ABB RobotStudio station: Solution14.rsstn

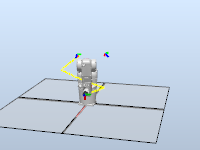
Station Solution14 (saved by RobotStudio 21.4.9700.0)
Controller IRB1200_7_70
  mechanical unit ROB_1: IRB1200_7_70_STD_03, 6 joints, base frame (0, 0, 0) mm
Layout (positions relative to the parent item):
  - IRB1200_7_70_STD_03 [mechanism, from Robots\IRB1200_7_70_STD_03.rslib] at (0, 0, 0) mm; joint values [0.2477, 0.9851, 0.7667, 0.2515, -1.7464, 0.0449] (rad or m)
Targets, tools, work objects and paths stored in the station, written as RAPID:
! task T_ROB1
MODULE Module1
  CONST robtarget Target_10:=[[422.01408311,0,750.1],[0.5,0,0.866025404,0],[0,0,0,0],[9E+09,9E+09,9E+09,9E+09,9E+09,9E+09]];
  CONST robtarget Target_20:=[[291.100367613,305.542897674,750.1],[0.459590616,-0.341070954,0.796034298,0.196917407],[0,0,-1,0],[9E+09,9E+09,9E+09,9E+09,9E+09,9E+09]];
  CONST jointtarget JointTarget_0:=[[-1.2,-19.89,29.46,-7.2,-9.64,7.1],[9E+09,9E+09,9E+09,9E+09,9E+09,9E+09]];
  CONST jointtarget JointTarget_1:=[[-2.4,-19.76,29.97,-13.32,-10.49,13.1],[9E+09,9E+09,9E+09,9E+09,9E+09,9E+09]];
  CONST jointtarget JointTarget_2:=[[-3.6,-19.59,30.47,-18.45,-11.45,18.1],[9E+09,9E+09,9E+09,9E+09,9E+09,9E+09]];
  CONST jointtarget JointTarget_3:=[[-4.79,-19.41,30.95,-22.74,-12.49,22.26],[9E+09,9E+09,9E+09,9E+09,9E+09,9E+09]];
  CONST jointtarget JointTarget_4:=[[-5.98,-19.2,31.42,-26.34,-13.59,25.69],[9E+09,9E+09,9E+09,9E+09,9E+09,9E+09]];
  CONST jointtarget JointTarget_5:=[[-7.17,-18.97,31.88,-29.36,-14.74,28.55],[9E+09,9E+09,9E+09,9E+09,9E+09,9E+09]];
  CONST jointtarget JointTarget_6:=[[-8.34,-18.72,32.33,-31.92,-15.92,30.93],[9E+09,9E+09,9E+09,9E+09,9E+09,9E+09]];
  CONST jointtarget JointTarget_7:=[[-9.51,-18.44,32.76,-34.11,-17.14,32.91],[9E+09,9E+09,9E+09,9E+09,9E+09,9E+09]];
  CONST jointtarget JointTarget_8:=[[-10.67,-18.14,33.17,-35.98,-18.37,34.57],[9E+09,9E+09,9E+09,9E+09,9E+09,9E+09]];
  CONST jointtarget JointTarget_9:=[[-11.82,-17.81,33.58,-37.61,-19.61,35.96],[9E+09,9E+09,9E+09,9E+09,9E+09,9E+09]];
  CONST jointtarget JointTarget_11:=[[-14.09,-17.09,34.33,-40.25,-22.13,38.1],[9E+09,9E+09,9E+09,9E+09,9E+09,9E+09]];
  CONST jointtarget JointTarget_12:=[[-15.21,-16.69,34.69,-41.34,-23.4,38.92],[9E+09,9E+09,9E+09,9E+09,9E+09,9E+09]];
  CONST jointtarget JointTarget_13:=[[-16.31,-16.27,35.03,-42.3,-24.66,39.59],[9E+09,9E+09,9E+09,9E+09,9E+09,9E+09]];
  CONST jointtarget JointTarget_14:=[[-17.4,-15.83,35.36,-43.16,-25.93,40.14],[9E+09,9E+09,9E+09,9E+09,9E+09,9E+09]];
  CONST jointtarget JointTarget_15:=[[-18.48,-15.37,35.67,-43.93,-27.19,40.6],[9E+09,9E+09,9E+09,9E+09,9E+09,9E+09]];
  CONST jointtarget JointTarget_16:=[[-19.55,-14.89,35.97,-44.63,-28.44,40.95],[9E+09,9E+09,9E+09,9E+09,9E+09,9E+09]];
  CONST jointtarget JointTarget_17:=[[-20.59,-14.38,36.24,-45.25,-29.69,41.23],[9E+09,9E+09,9E+09,9E+09,9E+09,9E+09]];
  CONST jointtarget JointTarget_18:=[[-21.63,-13.85,36.51,-45.83,-30.92,41.44],[9E+09,9E+09,9E+09,9E+09,9E+09,9E+09]];
  CONST jointtarget JointTarget_19:=[[-22.65,-13.3,36.75,-46.35,-32.15,41.59],[9E+09,9E+09,9E+09,9E+09,9E+09,9E+09]];
  CONST jointtarget JointTarget_21:=[[-24.64,-12.14,37.2,-47.28,-34.58,41.72],[9E+09,9E+09,9E+09,9E+09,9E+09,9E+09]];
  CONST jointtarget JointTarget_22:=[[-25.61,-11.53,37.4,-47.7,-35.77,41.72],[9E+09,9E+09,9E+09,9E+09,9E+09,9E+09]];
  CONST jointtarget JointTarget_23:=[[-26.57,-10.9,37.58,-48.09,-36.95,41.68],[9E+09,9E+09,9E+09,9E+09,9E+09,9E+09]];
  CONST jointtarget JointTarget_24:=[[-27.51,-10.26,37.74,-48.45,-38.11,41.6],[9E+09,9E+09,9E+09,9E+09,9E+09,9E+09]];
  CONST jointtarget JointTarget_25:=[[-28.43,-9.59,37.89,-48.8,-39.26,41.49],[9E+09,9E+09,9E+09,9E+09,9E+09,9E+09]];
  CONST jointtarget JointTarget_26:=[[-29.34,-8.91,38.02,-49.13,-40.39,41.35],[9E+09,9E+09,9E+09,9E+09,9E+09,9E+09]];
  CONST jointtarget JointTarget_27:=[[-30.23,-8.21,38.13,-49.44,-41.51,41.19],[9E+09,9E+09,9E+09,9E+09,9E+09,9E+09]];
  CONST jointtarget JointTarget_28:=[[-31.1,-7.5,38.22,-49.74,-42.6,41],[9E+09,9E+09,9E+09,9E+09,9E+09,9E+09]];
  CONST jointtarget JointTarget_29:=[[-31.96,-6.77,38.3,-50.03,-43.68,40.79],[9E+09,9E+09,9E+09,9E+09,9E+09,9E+09]];
  CONST jointtarget JointTarget_30:=[[-32.8,-6.03,38.36,-50.32,-44.75,40.56],[9E+09,9E+09,9E+09,9E+09,9E+09,9E+09]];
  CONST jointtarget JointTarget_31:=[[-33.63,-5.27,38.4,-50.59,-45.79,40.32],[9E+09,9E+09,9E+09,9E+09,9E+09,9E+09]];
  CONST jointtarget JointTarget_32:=[[-34.44,-4.51,38.43,-50.86,-46.82,40.06],[9E+09,9E+09,9E+09,9E+09,9E+09,9E+09]];
  CONST jointtarget JointTarget_33:=[[-35.23,-3.73,38.44,-51.12,-47.82,39.79],[9E+09,9E+09,9E+09,9E+09,9E+09,9E+09]];
  CONST jointtarget JointTarget_34:=[[-36.01,-2.93,38.43,-51.38,-48.81,39.5],[9E+09,9E+09,9E+09,9E+09,9E+09,9E+09]];
  CONST jointtarget JointTarget_35:=[[-36.77,-2.13,38.4,-51.64,-49.77,39.21],[9E+09,9E+09,9E+09,9E+09,9E+09,9E+09]];
  CONST jointtarget JointTarget_36:=[[-37.52,-1.32,38.36,-51.89,-50.72,38.91],[9E+09,9E+09,9E+09,9E+09,9E+09,9E+09]];
  CONST jointtarget JointTarget_37:=[[-38.25,-0.5,38.29,-52.14,-51.65,38.6],[9E+09,9E+09,9E+09,9E+09,9E+09,9E+09]];
  CONST jointtarget JointTarget_38:=[[-38.97,0.33,38.22,-52.39,-52.55,38.28],[9E+09,9E+09,9E+09,9E+09,9E+09,9E+09]];
  CONST jointtarget JointTarget_39:=[[-39.67,1.17,38.12,-52.64,-53.44,37.96],[9E+09,9E+09,9E+09,9E+09,9E+09,9E+09]];
  CONST jointtarget JointTarget_40:=[[-40.36,2.02,38,-52.89,-54.3,37.64],[9E+09,9E+09,9E+09,9E+09,9E+09,9E+09]];
  CONST jointtarget JointTarget_41:=[[-41.03,2.87,37.87,-53.14,-55.14,37.31],[9E+09,9E+09,9E+09,9E+09,9E+09,9E+09]];
  CONST jointtarget JointTarget_42:=[[-41.69,3.72,37.72,-53.38,-55.96,36.99],[9E+09,9E+09,9E+09,9E+09,9E+09,9E+09]];
  CONST jointtarget JointTarget_43:=[[-42.34,4.59,37.56,-53.63,-56.77,36.66],[9E+09,9E+09,9E+09,9E+09,9E+09,9E+09]];
  CONST jointtarget JointTarget_44:=[[-42.97,5.45,37.38,-53.88,-57.55,36.33],[9E+09,9E+09,9E+09,9E+09,9E+09,9E+09]];
  CONST jointtarget JointTarget_45:=[[-43.59,6.32,37.18,-54.13,-58.31,36],[9E+09,9E+09,9E+09,9E+09,9E+09,9E+09]];
  CONST jointtarget JointTarget_46:=[[-44.2,7.19,36.96,-54.38,-59.05,35.68],[9E+09,9E+09,9E+09,9E+09,9E+09,9E+09]];
  CONST jointtarget JointTarget_47:=[[-44.79,8.07,36.73,-54.64,-59.76,35.36],[9E+09,9E+09,9E+09,9E+09,9E+09,9E+09]];
  CONST jointtarget JointTarget_48:=[[-45.38,8.95,36.48,-54.89,-60.46,35.04],[9E+09,9E+09,9E+09,9E+09,9E+09,9E+09]];
  CONST jointtarget JointTarget_49:=[[-45.95,9.83,36.22,-55.14,-61.14,34.72],[9E+09,9E+09,9E+09,9E+09,9E+09,9E+09]];
  CONST jointtarget JointTarget_50:=[[-45.2,9.58,37.02,-54.18,-61.05,33.86],[9E+09,9E+09,9E+09,9E+09,9E+09,9E+09]];
  CONST jointtarget JointTarget_51:=[[-44.43,9.35,37.81,-53.2,-60.95,32.99],[9E+09,9E+09,9E+09,9E+09,9E+09,9E+09]];
  CONST jointtarget JointTarget_52:=[[-43.63,9.12,38.59,-52.19,-60.86,32.11],[9E+09,9E+09,9E+09,9E+09,9E+09,9E+09]];
  CONST jointtarget JointTarget_53:=[[-42.82,8.91,39.36,-51.15,-60.78,31.22],[9E+09,9E+09,9E+09,9E+09,9E+09,9E+09]];
  CONST jointtarget JointTarget_54:=[[-41.98,8.72,40.12,-50.08,-60.7,30.32],[9E+09,9E+09,9E+09,9E+09,9E+09,9E+09]];
  CONST jointtarget JointTarget_55:=[[-41.12,8.53,40.86,-48.99,-60.64,29.41],[9E+09,9E+09,9E+09,9E+09,9E+09,9E+09]];
  CONST jointtarget JointTarget_56:=[[-40.24,8.36,41.59,-47.87,-60.59,28.5],[9E+09,9E+09,9E+09,9E+09,9E+09,9E+09]];
  CONST jointtarget JointTarget_57:=[[-39.33,8.21,42.31,-46.71,-60.54,27.57],[9E+09,9E+09,9E+09,9E+09,9E+09,9E+09]];
  CONST jointtarget JointTarget_58:=[[-38.4,8.07,43.02,-45.53,-60.51,26.63],[9E+09,9E+09,9E+09,9E+09,9E+09,9E+09]];
  CONST jointtarget JointTarget_59:=[[-37.45,7.95,43.71,-44.32,-60.49,25.69],[9E+09,9E+09,9E+09,9E+09,9E+09,9E+09]];
  CONST jointtarget JointTarget_60:=[[-36.47,7.84,44.39,-43.08,-60.49,24.73],[9E+09,9E+09,9E+09,9E+09,9E+09,9E+09]];
  CONST jointtarget JointTarget_61:=[[-35.46,7.76,45.05,-41.81,-60.5,23.76],[9E+09,9E+09,9E+09,9E+09,9E+09,9E+09]];
  CONST jointtarget JointTarget_62:=[[-34.43,7.68,45.7,-40.5,-60.53,22.79],[9E+09,9E+09,9E+09,9E+09,9E+09,9E+09]];
  CONST jointtarget JointTarget_63:=[[-33.38,7.63,46.33,-39.17,-60.58,21.81],[9E+09,9E+09,9E+09,9E+09,9E+09,9E+09]];
  CONST jointtarget JointTarget_64:=[[-32.29,7.6,46.95,-37.81,-60.64,20.83],[9E+09,9E+09,9E+09,9E+09,9E+09,9E+09]];
  CONST jointtarget JointTarget_65:=[[-31.18,7.58,47.55,-36.41,-60.72,19.84],[9E+09,9E+09,9E+09,9E+09,9E+09,9E+09]];
  CONST jointtarget JointTarget_66:=[[-30.05,7.59,48.14,-34.99,-60.83,18.84],[9E+09,9E+09,9E+09,9E+09,9E+09,9E+09]];
  CONST jointtarget JointTarget_67:=[[-28.88,7.62,48.71,-33.54,-60.95,17.84],[9E+09,9E+09,9E+09,9E+09,9E+09,9E+09]];
  CONST jointtarget JointTarget_68:=[[-27.69,7.66,49.26,-32.06,-61.1,16.84],[9E+09,9E+09,9E+09,9E+09,9E+09,9E+09]];
  CONST jointtarget JointTarget_69:=[[-26.48,7.73,49.79,-30.56,-61.27,15.84],[9E+09,9E+09,9E+09,9E+09,9E+09,9E+09]];
  CONST jointtarget JointTarget_70:=[[-25.24,7.82,50.3,-29.03,-61.47,14.85],[9E+09,9E+09,9E+09,9E+09,9E+09,9E+09]];
  CONST jointtarget JointTarget_71:=[[-23.97,7.94,50.8,-27.48,-61.69,13.85],[9E+09,9E+09,9E+09,9E+09,9E+09,9E+09]];
  CONST jointtarget JointTarget_72:=[[-22.67,8.07,51.28,-25.9,-61.94,12.87],[9E+09,9E+09,9E+09,9E+09,9E+09,9E+09]];
  CONST jointtarget JointTarget_73:=[[-21.35,8.24,51.73,-24.31,-62.21,11.89],[9E+09,9E+09,9E+09,9E+09,9E+09,9E+09]];
  CONST jointtarget JointTarget_74:=[[-20.01,8.42,52.16,-22.69,-62.52,10.92],[9E+09,9E+09,9E+09,9E+09,9E+09,9E+09]];
  CONST jointtarget JointTarget_75:=[[-18.65,8.63,52.58,-21.06,-62.84,9.97],[9E+09,9E+09,9E+09,9E+09,9E+09,9E+09]];
  CONST jointtarget JointTarget_76:=[[-17.26,8.86,52.97,-19.41,-63.2,9.03],[9E+09,9E+09,9E+09,9E+09,9E+09,9E+09]];
  CONST jointtarget JointTarget_77:=[[-15.85,9.12,53.33,-17.75,-63.58,8.11],[9E+09,9E+09,9E+09,9E+09,9E+09,9E+09]];
  CONST jointtarget JointTarget_78:=[[-14.42,9.4,53.68,-16.08,-63.99,7.21],[9E+09,9E+09,9E+09,9E+09,9E+09,9E+09]];
  CONST jointtarget JointTarget_79:=[[-12.97,9.7,54,-14.41,-64.42,6.33],[9E+09,9E+09,9E+09,9E+09,9E+09,9E+09]];
  CONST jointtarget JointTarget_80:=[[-11.5,10.03,54.3,-12.73,-64.88,5.48],[9E+09,9E+09,9E+09,9E+09,9E+09,9E+09]];
  CONST jointtarget JointTarget_81:=[[-10.02,10.38,54.57,-11.04,-65.36,4.65],[9E+09,9E+09,9E+09,9E+09,9E+09,9E+09]];
  CONST jointtarget JointTarget_82:=[[-8.53,10.76,54.81,-9.35,-65.86,3.85],[9E+09,9E+09,9E+09,9E+09,9E+09,9E+09]];
  CONST jointtarget JointTarget_83:=[[-7.02,11.15,55.03,-7.67,-66.37,3.09],[9E+09,9E+09,9E+09,9E+09,9E+09,9E+09]];
  CONST jointtarget JointTarget_84:=[[-5.51,11.57,55.23,-5.99,-66.91,2.36],[9E+09,9E+09,9E+09,9E+09,9E+09,9E+09]];
  CONST jointtarget JointTarget_85:=[[-3.98,12.01,55.39,-4.31,-67.46,1.66],[9E+09,9E+09,9E+09,9E+09,9E+09,9E+09]];
  CONST jointtarget JointTarget_86:=[[-2.45,12.47,55.53,-2.65,-68.02,0.99],[9E+09,9E+09,9E+09,9E+09,9E+09,9E+09]];
  CONST jointtarget JointTarget_87:=[[-0.92,12.95,55.64,-0.99,-68.6,0.36],[9E+09,9E+09,9E+09,9E+09,9E+09,9E+09]];
  CONST jointtarget JointTarget_88:=[[0.61,13.45,55.73,0.66,-69.18,-0.23],[9E+09,9E+09,9E+09,9E+09,9E+09,9E+09]];
  CONST jointtarget JointTarget_89:=[[2.15,13.96,55.79,2.29,-69.76,-0.79],[9E+09,9E+09,9E+09,9E+09,9E+09,9E+09]];
  CONST jointtarget JointTarget_90:=[[3.68,14.49,55.82,3.9,-70.35,-1.31],[9E+09,9E+09,9E+09,9E+09,9E+09,9E+09]];
  CONST jointtarget JointTarget_91:=[[5.2,15.03,55.82,5.5,-70.93,-1.8],[9E+09,9E+09,9E+09,9E+09,9E+09,9E+09]];
  CONST jointtarget JointTarget_92:=[[6.72,15.59,55.79,7.09,-71.52,-2.26],[9E+09,9E+09,9E+09,9E+09,9E+09,9E+09]];
  CONST jointtarget JointTarget_93:=[[8.23,16.16,55.74,8.65,-72.09,-2.68],[9E+09,9E+09,9E+09,9E+09,9E+09,9E+09]];
  CONST jointtarget JointTarget_94:=[[9.72,16.74,55.65,10.19,-72.66,-3.07],[9E+09,9E+09,9E+09,9E+09,9E+09,9E+09]];
  CONST jointtarget JointTarget_95:=[[11.21,17.33,55.54,11.71,-73.21,-3.43],[9E+09,9E+09,9E+09,9E+09,9E+09,9E+09]];
  CONST jointtarget JointTarget_96:=[[12.68,17.93,55.41,13.21,-73.76,-3.76],[9E+09,9E+09,9E+09,9E+09,9E+09,9E+09]];
  CONST jointtarget JointTarget_97:=[[14.13,18.54,55.24,14.69,-74.28,-4.06],[9E+09,9E+09,9E+09,9E+09,9E+09,9E+09]];
  CONST jointtarget JointTarget_98:=[[15.56,19.15,55.05,16.14,-74.79,-4.34],[9E+09,9E+09,9E+09,9E+09,9E+09,9E+09]];
  CONST jointtarget JointTarget_99:=[[16.97,19.76,54.84,17.57,-75.29,-4.6],[9E+09,9E+09,9E+09,9E+09,9E+09,9E+09]];
  CONST jointtarget JointTarget_100:=[[18.11,20.22,55.2,18.67,-76.16,-4.62],[9E+09,9E+09,9E+09,9E+09,9E+09,9E+09]];
  CONST jointtarget JointTarget_101:=[[19.26,20.69,55.54,19.79,-77.02,-4.62],[9E+09,9E+09,9E+09,9E+09,9E+09,9E+09]];
  CONST jointtarget JointTarget_102:=[[20.44,21.19,55.87,20.92,-77.88,-4.59],[9E+09,9E+09,9E+09,9E+09,9E+09,9E+09]];
  CONST jointtarget JointTarget_103:=[[21.63,21.7,56.18,22.07,-78.74,-4.53],[9E+09,9E+09,9E+09,9E+09,9E+09,9E+09]];
  CONST jointtarget JointTarget_104:=[[22.84,22.23,56.46,23.24,-79.59,-4.44],[9E+09,9E+09,9E+09,9E+09,9E+09,9E+09]];
  CONST jointtarget JointTarget_105:=[[24.06,22.77,56.73,24.42,-80.42,-4.32],[9E+09,9E+09,9E+09,9E+09,9E+09,9E+09]];
  CONST jointtarget JointTarget_106:=[[25.3,23.33,56.97,25.62,-81.25,-4.18],[9E+09,9E+09,9E+09,9E+09,9E+09,9E+09]];
  CONST jointtarget JointTarget_107:=[[26.56,23.91,57.2,26.84,-82.05,-4],[9E+09,9E+09,9E+09,9E+09,9E+09,9E+09]];
  CONST jointtarget JointTarget_108:=[[27.83,24.5,57.4,28.07,-82.84,-3.8],[9E+09,9E+09,9E+09,9E+09,9E+09,9E+09]];
  CONST jointtarget JointTarget_109:=[[29.12,25.1,57.59,29.32,-83.61,-3.57],[9E+09,9E+09,9E+09,9E+09,9E+09,9E+09]];
  CONST jointtarget JointTarget_110:=[[30.41,25.71,57.75,30.58,-84.36,-3.32],[9E+09,9E+09,9E+09,9E+09,9E+09,9E+09]];
  CONST jointtarget JointTarget_111:=[[31.72,26.33,57.88,31.85,-85.08,-3.05],[9E+09,9E+09,9E+09,9E+09,9E+09,9E+09]];
  CONST jointtarget JointTarget_112:=[[33.03,26.96,58,33.13,-85.78,-2.75],[9E+09,9E+09,9E+09,9E+09,9E+09,9E+09]];
  CONST jointtarget JointTarget_113:=[[34.36,27.6,58.1,34.43,-86.45,-2.43],[9E+09,9E+09,9E+09,9E+09,9E+09,9E+09]];
  CONST jointtarget JointTarget_114:=[[35.69,28.25,58.17,35.74,-87.09,-2.09],[9E+09,9E+09,9E+09,9E+09,9E+09,9E+09]];
  CONST jointtarget JointTarget_115:=[[37.02,28.9,58.21,37.06,-87.69,-1.74],[9E+09,9E+09,9E+09,9E+09,9E+09,9E+09]];
  CONST jointtarget JointTarget_116:=[[38.36,29.55,58.24,38.38,-88.27,-1.37],[9E+09,9E+09,9E+09,9E+09,9E+09,9E+09]];
  CONST jointtarget JointTarget_117:=[[39.71,30.2,58.24,39.72,-88.8,-0.99],[9E+09,9E+09,9E+09,9E+09,9E+09,9E+09]];
  CONST jointtarget JointTarget_118:=[[41.05,30.86,58.22,41.05,-89.31,-0.6],[9E+09,9E+09,9E+09,9E+09,9E+09,9E+09]];
  CONST jointtarget JointTarget_119:=[[42.39,31.52,58.18,42.39,-89.78,-0.21],[9E+09,9E+09,9E+09,9E+09,9E+09,9E+09]];
  CONST jointtarget JointTarget_120:=[[43.74,32.17,58.11,43.74,-90.21,0.2],[9E+09,9E+09,9E+09,9E+09,9E+09,9E+09]];
  CONST jointtarget JointTarget_121:=[[45.07,32.83,58.02,45.08,-90.6,0.6],[9E+09,9E+09,9E+09,9E+09,9E+09,9E+09]];
  CONST jointtarget JointTarget_122:=[[46.41,33.48,57.91,46.41,-90.96,1],[9E+09,9E+09,9E+09,9E+09,9E+09,9E+09]];
  CONST jointtarget JointTarget_123:=[[47.73,34.12,57.77,47.75,-91.28,1.4],[9E+09,9E+09,9E+09,9E+09,9E+09,9E+09]];
  CONST jointtarget JointTarget_124:=[[49.05,34.76,57.62,49.08,-91.56,1.8],[9E+09,9E+09,9E+09,9E+09,9E+09,9E+09]];
  CONST jointtarget JointTarget_125:=[[50.36,35.4,57.44,50.4,-91.81,2.19],[9E+09,9E+09,9E+09,9E+09,9E+09,9E+09]];
  CONST jointtarget JointTarget_126:=[[51.66,36.03,57.24,51.71,-92.02,2.56],[9E+09,9E+09,9E+09,9E+09,9E+09,9E+09]];
  CONST jointtarget JointTarget_127:=[[52.95,36.65,57.02,53.01,-92.21,2.93],[9E+09,9E+09,9E+09,9E+09,9E+09,9E+09]];
  CONST jointtarget JointTarget_128:=[[54.23,37.26,56.78,54.3,-92.36,3.28],[9E+09,9E+09,9E+09,9E+09,9E+09,9E+09]];
  CONST jointtarget JointTarget_129:=[[55.49,37.86,56.51,55.57,-92.48,3.61],[9E+09,9E+09,9E+09,9E+09,9E+09,9E+09]];
  CONST jointtarget JointTarget_130:=[[56.74,38.46,56.23,56.83,-92.57,3.92],[9E+09,9E+09,9E+09,9E+09,9E+09,9E+09]];
  CONST jointtarget JointTarget_131:=[[57.97,39.05,55.93,58.07,-92.64,4.22],[9E+09,9E+09,9E+09,9E+09,9E+09,9E+09]];
  CONST jointtarget JointTarget_132:=[[59.19,39.62,55.61,59.3,-92.68,4.5],[9E+09,9E+09,9E+09,9E+09,9E+09,9E+09]];
  CONST jointtarget JointTarget_133:=[[60.39,40.19,55.27,60.5,-92.7,4.75],[9E+09,9E+09,9E+09,9E+09,9E+09,9E+09]];
  CONST jointtarget JointTarget_134:=[[61.57,40.75,54.91,61.69,-92.69,4.98],[9E+09,9E+09,9E+09,9E+09,9E+09,9E+09]];
  CONST jointtarget JointTarget_135:=[[62.74,41.3,54.54,62.86,-92.67,5.19],[9E+09,9E+09,9E+09,9E+09,9E+09,9E+09]];
  CONST jointtarget JointTarget_136:=[[63.88,41.85,54.14,64,-92.63,5.38],[9E+09,9E+09,9E+09,9E+09,9E+09,9E+09]];
  CONST jointtarget JointTarget_137:=[[65.01,42.38,53.73,65.13,-92.58,5.54],[9E+09,9E+09,9E+09,9E+09,9E+09,9E+09]];
  CONST jointtarget JointTarget_138:=[[66.11,42.9,53.31,66.24,-92.51,5.68],[9E+09,9E+09,9E+09,9E+09,9E+09,9E+09]];
  CONST jointtarget JointTarget_139:=[[67.2,43.42,52.86,67.32,-92.43,5.8],[9E+09,9E+09,9E+09,9E+09,9E+09,9E+09]];
  CONST jointtarget JointTarget_140:=[[68.26,43.93,52.41,68.38,-92.34,5.89],[9E+09,9E+09,9E+09,9E+09,9E+09,9E+09]];
  CONST jointtarget JointTarget_141:=[[69.31,44.43,51.93,69.42,-92.24,5.96],[9E+09,9E+09,9E+09,9E+09,9E+09,9E+09]];
  CONST jointtarget JointTarget_142:=[[70.33,44.92,51.45,70.44,-92.14,6],[9E+09,9E+09,9E+09,9E+09,9E+09,9E+09]];
  CONST jointtarget JointTarget_143:=[[71.34,45.41,50.95,71.44,-92.03,6.02],[9E+09,9E+09,9E+09,9E+09,9E+09,9E+09]];
  CONST jointtarget JointTarget_144:=[[72.32,45.89,50.43,72.42,-91.92,6.02],[9E+09,9E+09,9E+09,9E+09,9E+09,9E+09]];
  CONST jointtarget JointTarget_145:=[[73.28,46.36,49.9,73.38,-91.8,6],[9E+09,9E+09,9E+09,9E+09,9E+09,9E+09]];
  CONST jointtarget JointTarget_146:=[[74.23,46.83,49.36,74.32,-91.68,5.96],[9E+09,9E+09,9E+09,9E+09,9E+09,9E+09]];
  CONST jointtarget JointTarget_147:=[[75.15,47.29,48.81,75.23,-91.56,5.89],[9E+09,9E+09,9E+09,9E+09,9E+09,9E+09]];
  CONST jointtarget JointTarget_148:=[[76.05,47.74,48.24,76.13,-91.44,5.81],[9E+09,9E+09,9E+09,9E+09,9E+09,9E+09]];
  CONST jointtarget JointTarget_149:=[[76.94,48.19,47.67,77,-91.32,5.71],[9E+09,9E+09,9E+09,9E+09,9E+09,9E+09]];
  CONST jointtarget JointTarget_150:=[[75.88,48.43,48.05,75.97,-91.58,6.28],[9E+09,9E+09,9E+09,9E+09,9E+09,9E+09]];
  CONST jointtarget JointTarget_151:=[[74.8,48.67,48.41,74.91,-91.85,6.84],[9E+09,9E+09,9E+09,9E+09,9E+09,9E+09]];
  CONST jointtarget JointTarget_152:=[[73.7,48.92,48.76,73.84,-92.15,7.37],[9E+09,9E+09,9E+09,9E+09,9E+09,9E+09]];
  CONST jointtarget JointTarget_153:=[[72.58,49.18,49.09,72.75,-92.47,7.89],[9E+09,9E+09,9E+09,9E+09,9E+09,9E+09]];
  CONST jointtarget JointTarget_154:=[[71.43,49.43,49.4,71.63,-92.8,8.38],[9E+09,9E+09,9E+09,9E+09,9E+09,9E+09]];
  CONST jointtarget JointTarget_155:=[[70.26,49.69,49.69,70.51,-93.16,8.84],[9E+09,9E+09,9E+09,9E+09,9E+09,9E+09]];
  CONST jointtarget JointTarget_156:=[[69.07,49.95,49.97,69.36,-93.53,9.28],[9E+09,9E+09,9E+09,9E+09,9E+09,9E+09]];
  CONST jointtarget JointTarget_157:=[[67.87,50.22,50.23,68.2,-93.92,9.69],[9E+09,9E+09,9E+09,9E+09,9E+09,9E+09]];
  CONST jointtarget JointTarget_158:=[[66.64,50.48,50.47,67.02,-94.32,10.07],[9E+09,9E+09,9E+09,9E+09,9E+09,9E+09]];
  CONST jointtarget JointTarget_159:=[[65.39,50.74,50.69,65.82,-94.74,10.42],[9E+09,9E+09,9E+09,9E+09,9E+09,9E+09]];
  CONST jointtarget JointTarget_160:=[[64.12,51.01,50.9,64.61,-95.16,10.74],[9E+09,9E+09,9E+09,9E+09,9E+09,9E+09]];
  CONST jointtarget JointTarget_161:=[[62.84,51.27,51.08,63.38,-95.6,11.02],[9E+09,9E+09,9E+09,9E+09,9E+09,9E+09]];
  CONST jointtarget JointTarget_162:=[[61.54,51.53,51.25,62.14,-96.05,11.27],[9E+09,9E+09,9E+09,9E+09,9E+09,9E+09]];
  CONST jointtarget JointTarget_163:=[[60.22,51.78,51.39,60.88,-96.5,11.48],[9E+09,9E+09,9E+09,9E+09,9E+09,9E+09]];
  CONST jointtarget JointTarget_164:=[[58.89,52.03,51.52,59.6,-96.95,11.66],[9E+09,9E+09,9E+09,9E+09,9E+09,9E+09]];
  CONST jointtarget JointTarget_165:=[[57.55,52.28,51.63,58.31,-97.41,11.8],[9E+09,9E+09,9E+09,9E+09,9E+09,9E+09]];
  CONST jointtarget JointTarget_166:=[[56.19,52.52,51.71,57.01,-97.86,11.9],[9E+09,9E+09,9E+09,9E+09,9E+09,9E+09]];
  CONST jointtarget JointTarget_167:=[[54.82,52.75,51.78,55.7,-98.31,11.96],[9E+09,9E+09,9E+09,9E+09,9E+09,9E+09]];
  CONST jointtarget JointTarget_168:=[[53.45,52.98,51.83,54.37,-98.75,11.99],[9E+09,9E+09,9E+09,9E+09,9E+09,9E+09]];
  CONST jointtarget JointTarget_169:=[[52.06,53.2,51.86,53.03,-99.19,11.98],[9E+09,9E+09,9E+09,9E+09,9E+09,9E+09]];
  CONST jointtarget JointTarget_170:=[[50.67,53.41,51.86,51.68,-99.61,11.93],[9E+09,9E+09,9E+09,9E+09,9E+09,9E+09]];
  CONST jointtarget JointTarget_171:=[[49.28,53.62,51.85,50.32,-100.02,11.84],[9E+09,9E+09,9E+09,9E+09,9E+09,9E+09]];
  CONST jointtarget JointTarget_172:=[[47.88,53.81,51.81,48.95,-100.41,11.72],[9E+09,9E+09,9E+09,9E+09,9E+09,9E+09]];
  CONST jointtarget JointTarget_173:=[[46.48,54,51.76,47.58,-100.78,11.57],[9E+09,9E+09,9E+09,9E+09,9E+09,9E+09]];
  CONST jointtarget JointTarget_174:=[[45.09,54.18,51.69,46.2,-101.13,11.38],[9E+09,9E+09,9E+09,9E+09,9E+09,9E+09]];
  CONST jointtarget JointTarget_175:=[[43.69,54.35,51.59,44.81,-101.45,11.16],[9E+09,9E+09,9E+09,9E+09,9E+09,9E+09]];
  CONST jointtarget JointTarget_176:=[[42.3,54.51,51.48,43.42,-101.75,10.91],[9E+09,9E+09,9E+09,9E+09,9E+09,9E+09]];
  CONST jointtarget JointTarget_177:=[[40.91,54.66,51.35,42.03,-102.03,10.64],[9E+09,9E+09,9E+09,9E+09,9E+09,9E+09]];
  CONST jointtarget JointTarget_178:=[[39.53,54.8,51.19,40.65,-102.27,10.34],[9E+09,9E+09,9E+09,9E+09,9E+09,9E+09]];
  CONST jointtarget JointTarget_179:=[[38.16,54.94,51.02,39.26,-102.48,10.02],[9E+09,9E+09,9E+09,9E+09,9E+09,9E+09]];
  CONST jointtarget JointTarget_180:=[[36.8,55.06,50.83,37.87,-102.66,9.68],[9E+09,9E+09,9E+09,9E+09,9E+09,9E+09]];
  CONST jointtarget JointTarget_181:=[[35.45,55.18,50.62,36.5,-102.81,9.32],[9E+09,9E+09,9E+09,9E+09,9E+09,9E+09]];
  CONST jointtarget JointTarget_182:=[[34.11,55.29,50.39,35.13,-102.93,8.94],[9E+09,9E+09,9E+09,9E+09,9E+09,9E+09]];
  CONST jointtarget JointTarget_183:=[[32.79,55.39,50.14,33.76,-103.01,8.56],[9E+09,9E+09,9E+09,9E+09,9E+09,9E+09]];
  CONST jointtarget JointTarget_184:=[[31.48,55.49,49.88,32.41,-103.06,8.16],[9E+09,9E+09,9E+09,9E+09,9E+09,9E+09]];
  CONST jointtarget JointTarget_185:=[[30.19,55.57,49.59,31.08,-103.07,7.76],[9E+09,9E+09,9E+09,9E+09,9E+09,9E+09]];
  CONST jointtarget JointTarget_186:=[[28.91,55.66,49.29,29.75,-103.05,7.35],[9E+09,9E+09,9E+09,9E+09,9E+09,9E+09]];
  CONST jointtarget JointTarget_187:=[[27.66,55.73,48.97,28.45,-103,6.95],[9E+09,9E+09,9E+09,9E+09,9E+09,9E+09]];
  CONST jointtarget JointTarget_188:=[[26.42,55.81,48.64,27.16,-102.91,6.54],[9E+09,9E+09,9E+09,9E+09,9E+09,9E+09]];
  CONST jointtarget JointTarget_189:=[[25.2,55.88,48.29,25.89,-102.79,6.13],[9E+09,9E+09,9E+09,9E+09,9E+09,9E+09]];
  CONST jointtarget JointTarget_190:=[[24,55.94,47.92,24.64,-102.64,5.73],[9E+09,9E+09,9E+09,9E+09,9E+09,9E+09]];
  CONST jointtarget JointTarget_191:=[[22.82,56,47.54,23.41,-102.46,5.34],[9E+09,9E+09,9E+09,9E+09,9E+09,9E+09]];
  CONST jointtarget JointTarget_192:=[[21.67,56.06,47.14,22.2,-102.25,4.95],[9E+09,9E+09,9E+09,9E+09,9E+09,9E+09]];
  CONST jointtarget JointTarget_193:=[[20.53,56.12,46.72,21.01,-102.01,4.57],[9E+09,9E+09,9E+09,9E+09,9E+09,9E+09]];
  CONST jointtarget JointTarget_194:=[[19.42,56.17,46.29,19.85,-101.74,4.2],[9E+09,9E+09,9E+09,9E+09,9E+09,9E+09]];
  CONST jointtarget JointTarget_195:=[[18.33,56.22,45.85,18.72,-101.45,3.85],[9E+09,9E+09,9E+09,9E+09,9E+09,9E+09]];
  CONST jointtarget JointTarget_196:=[[17.26,56.28,45.39,17.6,-101.14,3.51],[9E+09,9E+09,9E+09,9E+09,9E+09,9E+09]];
  CONST jointtarget JointTarget_197:=[[16.21,56.33,44.92,16.51,-100.8,3.18],[9E+09,9E+09,9E+09,9E+09,9E+09,9E+09]];
  CONST jointtarget JointTarget_198:=[[15.19,56.39,44.43,15.45,-100.44,2.87],[9E+09,9E+09,9E+09,9E+09,9E+09,9E+09]];
  CONST jointtarget JointTarget_199:=[[14.19,56.44,43.93,14.41,-100.06,2.57],[9E+09,9E+09,9E+09,9E+09,9E+09,9E+09]];
  CONST jointtarget JointTarget_20:=[[-23.65,-12.73,36.98,-46.84,-33.37,41.68],[9E+09,9E+09,9E+09,9E+09,9E+09,9E+09]];
  CONST jointtarget JointTarget_10:=[[-12.96,-17.46,33.96,-39.02,-20.87,37.13],[9E+09,9E+09,9E+09,9E+09,9E+09,9E+09]];
  PROC Path_10()
    MoveAbsJ JointTarget_0,v100,z1,tool0\WObj:=wobj0;
    MoveAbsJ JointTarget_1,v100,z1,tool0\WObj:=wobj0;
    MoveAbsJ JointTarget_2,v100,z1,tool0\WObj:=wobj0;
    MoveAbsJ JointTarget_3,v100,z1,tool0\WObj:=wobj0;
    MoveAbsJ JointTarget_4,v100,z1,tool0\WObj:=wobj0;
    MoveAbsJ JointTarget_5,v100,z1,tool0\WObj:=wobj0;
    MoveAbsJ JointTarget_6,v100,z1,tool0\WObj:=wobj0;
    MoveAbsJ JointTarget_7,v100,z1,tool0\WObj:=wobj0;
    MoveAbsJ JointTarget_8,v100,z1,tool0\WObj:=wobj0;
    MoveAbsJ JointTarget_9,v100,z1,tool0\WObj:=wobj0;
    MoveAbsJ JointTarget_10,v100,z1,tool0\WObj:=wobj0;
    MoveAbsJ JointTarget_11,v100,z1,tool0\WObj:=wobj0;
    MoveAbsJ JointTarget_12,v100,z1,tool0\WObj:=wobj0;
    MoveAbsJ JointTarget_13,v100,z1,tool0\WObj:=wobj0;
    MoveAbsJ JointTarget_14,v100,z1,tool0\WObj:=wobj0;
    MoveAbsJ JointTarget_15,v100,z1,tool0\WObj:=wobj0;
    MoveAbsJ JointTarget_16,v100,z1,tool0\WObj:=wobj0;
    MoveAbsJ JointTarget_17,v100,z1,tool0\WObj:=wobj0;
    MoveAbsJ JointTarget_18,v100,z1,tool0\WObj:=wobj0;
    MoveAbsJ JointTarget_19,v100,z1,tool0\WObj:=wobj0;
    MoveAbsJ JointTarget_20,v100,z1,tool0\WObj:=wobj0;
    MoveAbsJ JointTarget_21,v100,z1,tool0\WObj:=wobj0;
    MoveAbsJ JointTarget_22,v100,z1,tool0\WObj:=wobj0;
    MoveAbsJ JointTarget_23,v100,z1,tool0\WObj:=wobj0;
    MoveAbsJ JointTarget_24,v100,z1,tool0\WObj:=wobj0;
    MoveAbsJ JointTarget_25,v100,z1,tool0\WObj:=wobj0;
    MoveAbsJ JointTarget_26,v100,z1,tool0\WObj:=wobj0;
    MoveAbsJ JointTarget_27,v100,z1,tool0\WObj:=wobj0;
    MoveAbsJ JointTarget_28,v100,z1,tool0\WObj:=wobj0;
    MoveAbsJ JointTarget_29,v100,z1,tool0\WObj:=wobj0;
    MoveAbsJ JointTarget_30,v100,z1,tool0\WObj:=wobj0;
    MoveAbsJ JointTarget_31,v100,z1,tool0\WObj:=wobj0;
    MoveAbsJ JointTarget_32,v100,z1,tool0\WObj:=wobj0;
    MoveAbsJ JointTarget_33,v100,z1,tool0\WObj:=wobj0;
    MoveAbsJ JointTarget_34,v100,z1,tool0\WObj:=wobj0;
    MoveAbsJ JointTarget_35,v100,z1,tool0\WObj:=wobj0;
    MoveAbsJ JointTarget_36,v100,z1,tool0\WObj:=wobj0;
    MoveAbsJ JointTarget_37,v100,z1,tool0\WObj:=wobj0;
    MoveAbsJ JointTarget_38,v100,z1,tool0\WObj:=wobj0;
    MoveAbsJ JointTarget_39,v100,z1,tool0\WObj:=wobj0;
    MoveAbsJ JointTarget_40,v100,z1,tool0\WObj:=wobj0;
    MoveAbsJ JointTarget_41,v100,z1,tool0\WObj:=wobj0;
    MoveAbsJ JointTarget_42,v100,z1,tool0\WObj:=wobj0;
    MoveAbsJ JointTarget_43,v100,z1,tool0\WObj:=wobj0;
    MoveAbsJ JointTarget_44,v100,z1,tool0\WObj:=wobj0;
    MoveAbsJ JointTarget_45,v100,z1,tool0\WObj:=wobj0;
    MoveAbsJ JointTarget_46,v100,z1,tool0\WObj:=wobj0;
    MoveAbsJ JointTarget_47,v100,z1,tool0\WObj:=wobj0;
    MoveAbsJ JointTarget_48,v100,z1,tool0\WObj:=wobj0;
    MoveAbsJ JointTarget_49,v100,z1,tool0\WObj:=wobj0;
    MoveAbsJ JointTarget_50,v100,z1,tool0\WObj:=wobj0;
    MoveAbsJ JointTarget_51,v100,z1,tool0\WObj:=wobj0;
    MoveAbsJ JointTarget_52,v100,z1,tool0\WObj:=wobj0;
    MoveAbsJ JointTarget_53,v100,z1,tool0\WObj:=wobj0;
    MoveAbsJ JointTarget_54,v100,z1,tool0\WObj:=wobj0;
    MoveAbsJ JointTarget_55,v100,z1,tool0\WObj:=wobj0;
    MoveAbsJ JointTarget_56,v100,z1,tool0\WObj:=wobj0;
    MoveAbsJ JointTarget_57,v100,z1,tool0\WObj:=wobj0;
    MoveAbsJ JointTarget_58,v100,z1,tool0\WObj:=wobj0;
    MoveAbsJ JointTarget_59,v100,z1,tool0\WObj:=wobj0;
    MoveAbsJ JointTarget_60,v100,z1,tool0\WObj:=wobj0;
    MoveAbsJ JointTarget_61,v100,z1,tool0\WObj:=wobj0;
    MoveAbsJ JointTarget_62,v100,z1,tool0\WObj:=wobj0;
    MoveAbsJ JointTarget_63,v100,z1,tool0\WObj:=wobj0;
    MoveAbsJ JointTarget_64,v100,z1,tool0\WObj:=wobj0;
    MoveAbsJ JointTarget_65,v100,z1,tool0\WObj:=wobj0;
    MoveAbsJ JointTarget_66,v100,z1,tool0\WObj:=wobj0;
    MoveAbsJ JointTarget_67,v100,z1,tool0\WObj:=wobj0;
    MoveAbsJ JointTarget_68,v100,z1,tool0\WObj:=wobj0;
    MoveAbsJ JointTarget_69,v100,z1,tool0\WObj:=wobj0;
    MoveAbsJ JointTarget_70,v100,z1,tool0\WObj:=wobj0;
    MoveAbsJ JointTarget_71,v100,z1,tool0\WObj:=wobj0;
    MoveAbsJ JointTarget_72,v100,z1,tool0\WObj:=wobj0;
    MoveAbsJ JointTarget_73,v100,z1,tool0\WObj:=wobj0;
    MoveAbsJ JointTarget_74,v100,z1,tool0\WObj:=wobj0;
    MoveAbsJ JointTarget_75,v100,z1,tool0\WObj:=wobj0;
    MoveAbsJ JointTarget_76,v100,z1,tool0\WObj:=wobj0;
    MoveAbsJ JointTarget_77,v100,z1,tool0\WObj:=wobj0;
    MoveAbsJ JointTarget_78,v100,z1,tool0\WObj:=wobj0;
    MoveAbsJ JointTarget_79,v100,z1,tool0\WObj:=wobj0;
    MoveAbsJ JointTarget_80,v100,z1,tool0\WObj:=wobj0;
    MoveAbsJ JointTarget_81,v100,z1,tool0\WObj:=wobj0;
    MoveAbsJ JointTarget_82,v100,z1,tool0\WObj:=wobj0;
    MoveAbsJ JointTarget_83,v100,z1,tool0\WObj:=wobj0;
    MoveAbsJ JointTarget_84,v100,z1,tool0\WObj:=wobj0;
    MoveAbsJ JointTarget_85,v100,z1,tool0\WObj:=wobj0;
    MoveAbsJ JointTarget_86,v100,z1,tool0\WObj:=wobj0;
    MoveAbsJ JointTarget_87,v100,z1,tool0\WObj:=wobj0;
    MoveAbsJ JointTarget_88,v100,z1,tool0\WObj:=wobj0;
    MoveAbsJ JointTarget_89,v100,z1,tool0\WObj:=wobj0;
    MoveAbsJ JointTarget_90,v100,z1,tool0\WObj:=wobj0;
    MoveAbsJ JointTarget_91,v100,z1,tool0\WObj:=wobj0;
    MoveAbsJ JointTarget_92,v100,z1,tool0\WObj:=wobj0;
    MoveAbsJ JointTarget_93,v100,z1,tool0\WObj:=wobj0;
    MoveAbsJ JointTarget_94,v100,z1,tool0\WObj:=wobj0;
    MoveAbsJ JointTarget_95,v100,z1,tool0\WObj:=wobj0;
    MoveAbsJ JointTarget_96,v100,z1,tool0\WObj:=wobj0;
    MoveAbsJ JointTarget_97,v100,z1,tool0\WObj:=wobj0;
    MoveAbsJ JointTarget_98,v100,z1,tool0\WObj:=wobj0;
    MoveAbsJ JointTarget_99,v100,z1,tool0\WObj:=wobj0;
    MoveAbsJ JointTarget_100,v100,z1,tool0\WObj:=wobj0;
    MoveAbsJ JointTarget_101,v100,z1,tool0\WObj:=wobj0;
    MoveAbsJ JointTarget_102,v100,z1,tool0\WObj:=wobj0;
    MoveAbsJ JointTarget_103,v100,z1,tool0\WObj:=wobj0;
    MoveAbsJ JointTarget_104,v100,z1,tool0\WObj:=wobj0;
    MoveAbsJ JointTarget_105,v100,z1,tool0\WObj:=wobj0;
    MoveAbsJ JointTarget_106,v100,z1,tool0\WObj:=wobj0;
    MoveAbsJ JointTarget_107,v100,z1,tool0\WObj:=wobj0;
    MoveAbsJ JointTarget_108,v100,z1,tool0\WObj:=wobj0;
    MoveAbsJ JointTarget_109,v100,z1,tool0\WObj:=wobj0;
    MoveAbsJ JointTarget_110,v100,z1,tool0\WObj:=wobj0;
    MoveAbsJ JointTarget_111,v100,z1,tool0\WObj:=wobj0;
    MoveAbsJ JointTarget_112,v100,z1,tool0\WObj:=wobj0;
    MoveAbsJ JointTarget_113,v100,z1,tool0\WObj:=wobj0;
    MoveAbsJ JointTarget_114,v100,z1,tool0\WObj:=wobj0;
    MoveAbsJ JointTarget_115,v100,z1,tool0\WObj:=wobj0;
    MoveAbsJ JointTarget_116,v100,z1,tool0\WObj:=wobj0;
    MoveAbsJ JointTarget_117,v100,z1,tool0\WObj:=wobj0;
    MoveAbsJ JointTarget_118,v100,z1,tool0\WObj:=wobj0;
    MoveAbsJ JointTarget_119,v100,z1,tool0\WObj:=wobj0;
    MoveAbsJ JointTarget_120,v100,z1,tool0\WObj:=wobj0;
    MoveAbsJ JointTarget_121,v100,z1,tool0\WObj:=wobj0;
    MoveAbsJ JointTarget_122,v100,z1,tool0\WObj:=wobj0;
    MoveAbsJ JointTarget_123,v100,z1,tool0\WObj:=wobj0;
    MoveAbsJ JointTarget_124,v100,z1,tool0\WObj:=wobj0;
    MoveAbsJ JointTarget_125,v100,z1,tool0\WObj:=wobj0;
    MoveAbsJ JointTarget_126,v100,z1,tool0\WObj:=wobj0;
    MoveAbsJ JointTarget_127,v100,z1,tool0\WObj:=wobj0;
    MoveAbsJ JointTarget_128,v100,z1,tool0\WObj:=wobj0;
    MoveAbsJ JointTarget_129,v100,z1,tool0\WObj:=wobj0;
    MoveAbsJ JointTarget_130,v100,z1,tool0\WObj:=wobj0;
    MoveAbsJ JointTarget_131,v100,z1,tool0\WObj:=wobj0;
    MoveAbsJ JointTarget_132,v100,z1,tool0\WObj:=wobj0;
    MoveAbsJ JointTarget_133,v100,z1,tool0\WObj:=wobj0;
    MoveAbsJ JointTarget_134,v100,z1,tool0\WObj:=wobj0;
    MoveAbsJ JointTarget_135,v100,z1,tool0\WObj:=wobj0;
    MoveAbsJ JointTarget_136,v100,z1,tool0\WObj:=wobj0;
    MoveAbsJ JointTarget_137,v100,z1,tool0\WObj:=wobj0;
    MoveAbsJ JointTarget_138,v100,z1,tool0\WObj:=wobj0;
    MoveAbsJ JointTarget_139,v100,z1,tool0\WObj:=wobj0;
    MoveAbsJ JointTarget_140,v100,z1,tool0\WObj:=wobj0;
    MoveAbsJ JointTarget_141,v100,z1,tool0\WObj:=wobj0;
    MoveAbsJ JointTarget_142,v100,z1,tool0\WObj:=wobj0;
    MoveAbsJ JointTarget_143,v100,z1,tool0\WObj:=wobj0;
    MoveAbsJ JointTarget_144,v100,z1,tool0\WObj:=wobj0;
    MoveAbsJ JointTarget_145,v100,z1,tool0\WObj:=wobj0;
    MoveAbsJ JointTarget_146,v100,z1,tool0\WObj:=wobj0;
    MoveAbsJ JointTarget_147,v100,z1,tool0\WObj:=wobj0;
    MoveAbsJ JointTarget_148,v100,z1,tool0\WObj:=wobj0;
    MoveAbsJ JointTarget_149,v100,z1,tool0\WObj:=wobj0;
    MoveAbsJ JointTarget_150,v100,z1,tool0\WObj:=wobj0;
    MoveAbsJ JointTarget_151,v100,z1,tool0\WObj:=wobj0;
    MoveAbsJ JointTarget_152,v100,z1,tool0\WObj:=wobj0;
    MoveAbsJ JointTarget_153,v100,z1,tool0\WObj:=wobj0;
    MoveAbsJ JointTarget_154,v100,z1,tool0\WObj:=wobj0;
    MoveAbsJ JointTarget_155,v100,z1,tool0\WObj:=wobj0;
    MoveAbsJ JointTarget_156,v100,z1,tool0\WObj:=wobj0;
    MoveAbsJ JointTarget_157,v100,z1,tool0\WObj:=wobj0;
    MoveAbsJ JointTarget_158,v100,z1,tool0\WObj:=wobj0;
    MoveAbsJ JointTarget_159,v100,z1,tool0\WObj:=wobj0;
    MoveAbsJ JointTarget_160,v100,z1,tool0\WObj:=wobj0;
    MoveAbsJ JointTarget_161,v100,z1,tool0\WObj:=wobj0;
    MoveAbsJ JointTarget_162,v100,z1,tool0\WObj:=wobj0;
    MoveAbsJ JointTarget_163,v100,z1,tool0\WObj:=wobj0;
    MoveAbsJ JointTarget_164,v100,z1,tool0\WObj:=wobj0;
    MoveAbsJ JointTarget_165,v100,z1,tool0\WObj:=wobj0;
    MoveAbsJ JointTarget_166,v100,z1,tool0\WObj:=wobj0;
    MoveAbsJ JointTarget_167,v100,z1,tool0\WObj:=wobj0;
    MoveAbsJ JointTarget_168,v100,z1,tool0\WObj:=wobj0;
    MoveAbsJ JointTarget_169,v100,z1,tool0\WObj:=wobj0;
    MoveAbsJ JointTarget_170,v100,z1,tool0\WObj:=wobj0;
    MoveAbsJ JointTarget_171,v100,z1,tool0\WObj:=wobj0;
    MoveAbsJ JointTarget_172,v100,z1,tool0\WObj:=wobj0;
    MoveAbsJ JointTarget_173,v100,z1,tool0\WObj:=wobj0;
    MoveAbsJ JointTarget_174,v100,z1,tool0\WObj:=wobj0;
    MoveAbsJ JointTarget_175,v100,z1,tool0\WObj:=wobj0;
    MoveAbsJ JointTarget_176,v100,z1,tool0\WObj:=wobj0;
    MoveAbsJ JointTarget_177,v100,z1,tool0\WObj:=wobj0;
    MoveAbsJ JointTarget_178,v100,z1,tool0\WObj:=wobj0;
    MoveAbsJ JointTarget_179,v100,z1,tool0\WObj:=wobj0;
    MoveAbsJ JointTarget_180,v100,z1,tool0\WObj:=wobj0;
    MoveAbsJ JointTarget_181,v100,z1,tool0\WObj:=wobj0;
    MoveAbsJ JointTarget_182,v100,z1,tool0\WObj:=wobj0;
    MoveAbsJ JointTarget_183,v100,z1,tool0\WObj:=wobj0;
    MoveAbsJ JointTarget_184,v100,z1,tool0\WObj:=wobj0;
    MoveAbsJ JointTarget_185,v100,z1,tool0\WObj:=wobj0;
    MoveAbsJ JointTarget_186,v100,z1,tool0\WObj:=wobj0;
    MoveAbsJ JointTarget_187,v100,z1,tool0\WObj:=wobj0;
    MoveAbsJ JointTarget_188,v100,z1,tool0\WObj:=wobj0;
    MoveAbsJ JointTarget_189,v100,z1,tool0\WObj:=wobj0;
    MoveAbsJ JointTarget_190,v100,z1,tool0\WObj:=wobj0;
    MoveAbsJ JointTarget_191,v100,z1,tool0\WObj:=wobj0;
    MoveAbsJ JointTarget_192,v100,z1,tool0\WObj:=wobj0;
    MoveAbsJ JointTarget_193,v100,z1,tool0\WObj:=wobj0;
    MoveAbsJ JointTarget_194,v100,z1,tool0\WObj:=wobj0;
    MoveAbsJ JointTarget_195,v100,z1,tool0\WObj:=wobj0;
    MoveAbsJ JointTarget_196,v100,z1,tool0\WObj:=wobj0;
    MoveAbsJ JointTarget_197,v100,z1,tool0\WObj:=wobj0;
    MoveAbsJ JointTarget_198,v100,z1,tool0\WObj:=wobj0;
    MoveAbsJ JointTarget_199,v100,z1,tool0\WObj:=wobj0;
  ENDPROC
  PROC main()
    Path_10;
  ENDPROC
ENDMODULE

